SYSTEM HiddenConnectionTest
  (* Version 1.0, 2022-03-29, LukasWais *)
  APPLICATION HiddenConnectionTestApp
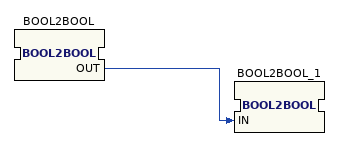
    FBS
      BOOL2BOOL : BOOL2BOOL;
      BOOL2BOOL_1 : BOOL2BOOL;
    END_FBS
    DATA_CONNECTIONS
      BOOL2BOOL.OUT TO BOOL2BOOL_1.IN;
    END_CONNECTIONS
  END_APPLICATION
END_SYSTEM
